FUNCTION_BLOCK Detector_N_Drawer (* Basic FB with empty ECC *)
  (* Standard: 61499-2 *)
  (* Version 1.0, 2024-11-25, obotnar *)
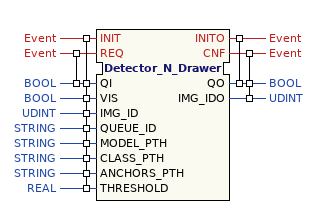
  EVENT_INPUT
    INIT WITH VIS, IMG_ID, QUEUE_ID, MODEL_PTH, CLASS_PTH, THRESHOLD, QI, ANCHORS_PTH;
    REQ WITH QI;
  END_EVENT
  EVENT_OUTPUT
    INITO WITH QO;
    CNF WITH QO, IMG_IDO;
  END_EVENT
  VAR_INPUT
    QI : BOOL;
    VIS : BOOL;
    IMG_ID : UDINT;
    QUEUE_ID : STRING;
    MODEL_PTH : STRING;
    CLASS_PTH : STRING;
    ANCHORS_PTH : STRING;
    THRESHOLD : REAL;
  END_VAR
  VAR_OUTPUT
    QO : BOOL;
    IMG_IDO : UDINT;
  END_VAR
  EC_STATES
    START; (* Initial State *)
  END_STATES
END_FUNCTION_BLOCK
